// TIA Portal V19 export
FUNCTION "FC_EM_Transport" : Void   // FC6, FBD
{ S7_Optimized_Access := 'TRUE' }
// stored: SetENOAutomatically false
BEGIN

REGION Network 1: ------------------------------------------------------------------------ Inputs ------------------------------------------------------------------------
END_REGION

REGION Network 2: Verwerking iTransportSenDown_h1
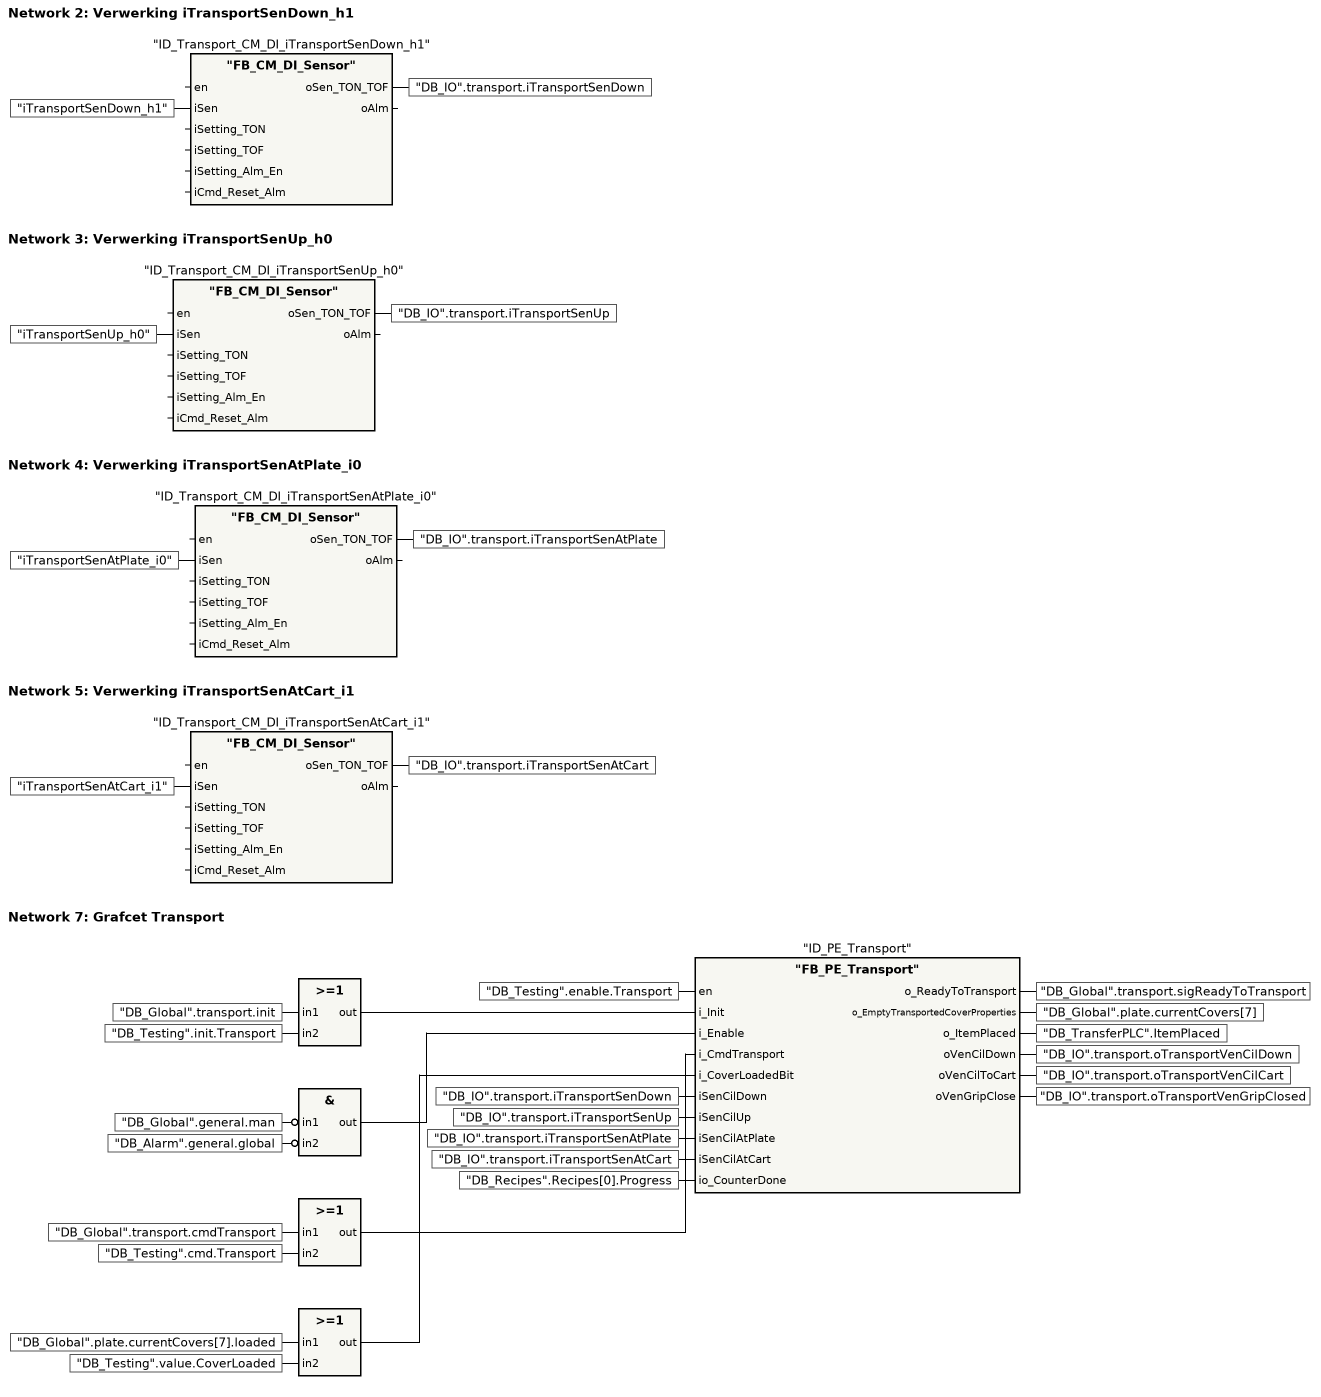
   "ID_Transport_CM_DI_iTransportSenDown_h1"(iSen := "iTransportSenDown_h1",   // "FB_CM_DI_Sensor"
                           oSen_TON_TOF => "DB_IO".transport.iTransportSenDown);
END_REGION

REGION Network 3: Verwerking iTransportSenUp_h0
   "ID_Transport_CM_DI_iTransportSenUp_h0"(iSen := "iTransportSenUp_h0",   // "FB_CM_DI_Sensor"
                           oSen_TON_TOF => "DB_IO".transport.iTransportSenUp);
END_REGION

REGION Network 4: Verwerking iTransportSenAtPlate_i0
   "ID_Transport_CM_DI_iTransportSenAtPlate_i0"(iSen := "iTransportSenAtPlate_i0",   // "FB_CM_DI_Sensor"
                           oSen_TON_TOF => "DB_IO".transport.iTransportSenAtPlate);
END_REGION

REGION Network 5: Verwerking iTransportSenAtCart_i1
   "ID_Transport_CM_DI_iTransportSenAtCart_i1"(iSen := "iTransportSenAtCart_i1",   // "FB_CM_DI_Sensor"
                           oSen_TON_TOF => "DB_IO".transport.iTransportSenAtCart);
END_REGION

REGION Network 6: ------------------------------------------------------------------------ Logic ------------------------------------------------------------------------
END_REGION

REGION Network 7: Grafcet Transport
   IF "DB_Testing".enable.Transport THEN
       "ID_PE_Transport"(i_Init := "DB_Global".transport.init OR "DB_Testing".init.Transport,   // "FB_PE_Transport"
                         i_Enable := NOT "DB_Global".general.man AND NOT "DB_Alarm".general.global,
                         i_CmdTransport := "DB_Global".transport.cmdTransport OR "DB_Testing".cmd.Transport,
                         i_CoverLoadedBit := "DB_Global".plate.currentCovers[7].loaded OR "DB_Testing".value.CoverLoaded,
                         iSenCilDown := "DB_IO".transport.iTransportSenDown,
                         iSenCilUp := "DB_IO".transport.iTransportSenUp,
                         iSenCilAtPlate := "DB_IO".transport.iTransportSenAtPlate,
                         iSenCilAtCart := "DB_IO".transport.iTransportSenAtCart,
                         io_CounterDone := "DB_Recipes".Recipes[0].Progress,
                         o_ReadyToTransport => "DB_Global".transport.sigReadyToTransport,
                         o_EmptyTransportedCoverProperties => "DB_Global".plate.currentCovers[7],
                         o_ItemPlaced => "DB_TransferPLC".ItemPlaced,
                         oVenCilDown => "DB_IO".transport.oTransportVenCilDown,
                         oVenCilToCart => "DB_IO".transport.oTransportVenCilCart,
                         oVenGripClose => "DB_IO".transport.oTransportVenGripClosed);
   END_IF;
END_REGION

REGION Network 8: ------------------------------------------------------------------------ Outputs ------------------------------------------------------------------------
END_REGION

REGION Network 9: Sturen oTransportVenCilDown_A+
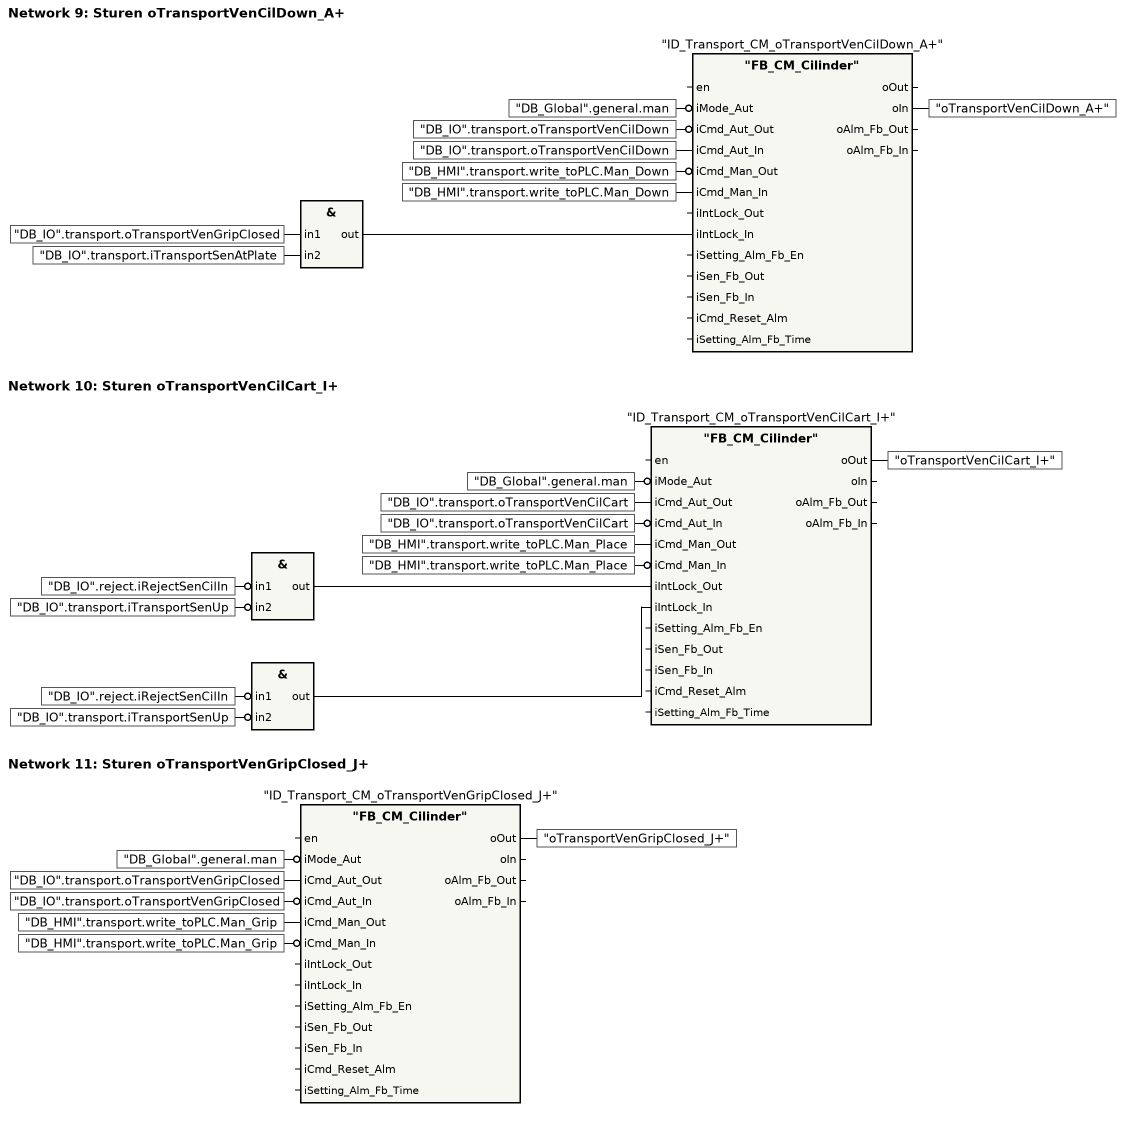
   "ID_Transport_CM_oTransportVenCilDown_A+"(iMode_Aut := NOT "DB_Global".general.man,   // "FB_CM_Cilinder"
                           iCmd_Aut_Out := NOT "DB_IO".transport.oTransportVenCilDown,
                           iCmd_Aut_In := "DB_IO".transport.oTransportVenCilDown,
                           iCmd_Man_Out := NOT "DB_HMI".transport.write_toPLC.Man_Down,
                           iCmd_Man_In := "DB_HMI".transport.write_toPLC.Man_Down,
                           iIntLock_In := "DB_IO".transport.oTransportVenGripClosed AND "DB_IO".transport.iTransportSenAtPlate,
                           oIn => "oTransportVenCilDown_A+");
END_REGION

REGION Network 10: Sturen oTransportVenCilCart_I+
   // TODO:
   // - Interlocks
   "ID_Transport_CM_oTransportVenCilCart_I+"(iMode_Aut := NOT "DB_Global".general.man,   // "FB_CM_Cilinder"
                           iCmd_Aut_Out := "DB_IO".transport.oTransportVenCilCart,
                           iCmd_Aut_In := NOT "DB_IO".transport.oTransportVenCilCart,
                           iCmd_Man_Out := "DB_HMI".transport.write_toPLC.Man_Place,
                           iCmd_Man_In := NOT "DB_HMI".transport.write_toPLC.Man_Place,
                           iIntLock_Out := NOT "DB_IO".reject.iRejectSenCilIn AND NOT "DB_IO".transport.iTransportSenUp,
                           iIntLock_In := NOT "DB_IO".reject.iRejectSenCilIn AND NOT "DB_IO".transport.iTransportSenUp,
                           oOut => "oTransportVenCilCart_I+");
END_REGION

REGION Network 11: Sturen oTransportVenGripClosed_J+
   "ID_Transport_CM_oTransportVenGripClosed_J+"(iMode_Aut := NOT "DB_Global".general.man,   // "FB_CM_Cilinder"
                           iCmd_Aut_Out := "DB_IO".transport.oTransportVenGripClosed,
                           iCmd_Aut_In := NOT "DB_IO".transport.oTransportVenGripClosed,
                           iCmd_Man_Out := "DB_HMI".transport.write_toPLC.Man_Grip,
                           iCmd_Man_In := NOT "DB_HMI".transport.write_toPLC.Man_Grip,
                           oOut => "oTransportVenGripClosed_J+");
END_REGION
END_FUNCTION
